// TIA Portal V19 export
TYPE "LAF_typeGeneralStatus"
TITLE = LAF_typeGeneralStatus
// Information of the general status of the unit
// stored: Access Published
   STRUCT
      acknowledge : Bool;   // Global acknowledge
      disableAlarms : Bool;   // Global command to disable all alarms
      activateSimulation : Bool;   // Set everything in simulation
      enablePower : Bool;   // Release to turn on power (e.g. 240V, contactors, drives)
      localPlcDateAndTime { ExternalWritable := 'False'} : "LAF_typeGlobalDateTime";   // Local date and time of the PLC
      dayLightSavingTime : Bool;   // Daylight saving time
      clock { ExternalWritable := 'False'} : "LAF_typeGlobalClockMem";
      posPulse { ExternalWritable := 'False'} : "LAF_typeGlobalClockMem";   // Positive pulse clock memory
      clockMemoryByte { ExternalWritable := 'False'} : Byte;   // Summarized clock bits in one byte
      firstCycle { ExternalWritable := 'False'} : Bool := true;   // First cycle of the CPU
   END_STRUCT;
END_TYPE
